FUNCTION_BLOCK XtsTrackStub IMPLEMENTS I_XtsTrack
VAR_INPUT
END_VAR
VAR_OUTPUT
END_VAR
VAR
	_trackLength : MC_LREAL  := 1000;
END_VAR

{warning 'add property implementation'}
PROPERTY MyOTCID : OTCID
GET
END_GET
SET
END_SET
END_PROPERTY

{warning 'add property implementation'}
PROPERTY TrackLength : MC_Lreal
GET
tracklength := _trackLength;
END_GET
END_PROPERTY

END_FUNCTION_BLOCK

(* stored: Version 1.1.0.1, ProductVersion 3.1.4024.12
   POU XtsTrackStub: Id {03c15466-6090-4765-816b-ccda66b9b333}, SpecialFunc None
   Property MyOTCID: Id {58d1505c-0536-4521-b091-1fd2d7ec90a0}
   Get Get: Id {942d4dc2-14a4-4bef-a1f1-3c53554951f2}
   Set Set: Id {3cae8b1f-6357-4ce3-be2f-9aa0e3e4f6bb}
   Property TrackLength: Id {6b606c91-c693-4cef-8de3-8222ee49a6d2}
   Get Get: Id {2e912149-8443-4ed1-8754-35c8863e5c66} *)
